TYPE TaskBaseInternal :
STRUCT
	_state : UDINT;
	_newCommand : BOOL;
	_activeCommand : IPLCOpenCommand;
END_STRUCT
END_TYPE

(* stored: Version 1.1.0.1
   DUT TaskBaseInternal: Id {c731ea55-51d4-436c-b5c4-ed556ae77e87} *)
